DATA_BLOCK "PENEIRAS_DB"
{ S7_Optimized_Access := 'TRUE' }
VERSION : 0.1
NON_RETAIN
"PENEIRAS"

BEGIN

END_DATA_BLOCK

